// TIA Portal V18 export
DATA_BLOCK "mixer"   // DB74
{ S7_Optimized_Access := 'TRUE' }
VERSION : 0.1
// stored: AutoNumber true, DBAccessibleFromOPCUA true, IsOnlyStoredInLoadMemory false, IsRetainMemResEnabled false, IsWriteProtectedInAS false, MemoryReserve 100
   VAR RETAIN
      "mixer enable" : Int;
      "mixer control enable" : Int;
   END_VAR
   VAR
      "mixer enabled" : Bool;
      "mixer control enabled" : Bool;
   END_VAR
   VAR RETAIN
      "mixer speed at20 mA" : Real;
      "mixer Speed maximum" : Real;
      "mixer speed" : Real;
   END_VAR
   VAR
      "mixer control time" : Int;
   END_VAR
BEGIN
END_DATA_BLOCK
